FUNCTION_BLOCK ProductOrders (* Basic Function Block Type *)
  (* Standard: 61499-2 *)
  (* Version 0.0, 5/28/2018, taavi, nxtControl GmbH, Template *)
  PACKAGE Main;
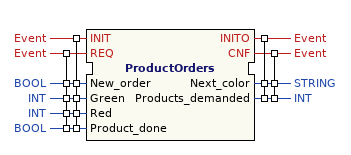
  EVENT_INPUT
    INIT WITH New_order, Green, Red, Product_done; (* Initialization Request *)
    REQ WITH Green, New_order, Product_done, Red; (* Normal Execution Request *)
  END_EVENT
  EVENT_OUTPUT
    INITO WITH Next_color, Products_demanded; (* Initialization Confirm *)
    CNF WITH Next_color, Products_demanded; (* Execution Confirmation *)
  END_EVENT
  VAR_INPUT
    New_order : BOOL;
    Green : INT; (* Input event qualifier *)
    Red : INT;
    Product_done : BOOL;
  END_VAR
  VAR_OUTPUT
    Next_color : STRING; (* Output event qualifier *)
    Products_demanded : INT;
  END_VAR
  VAR
    Green_count : INT;
    Red_count : INT;
    Product_count : INT;
  END_VAR
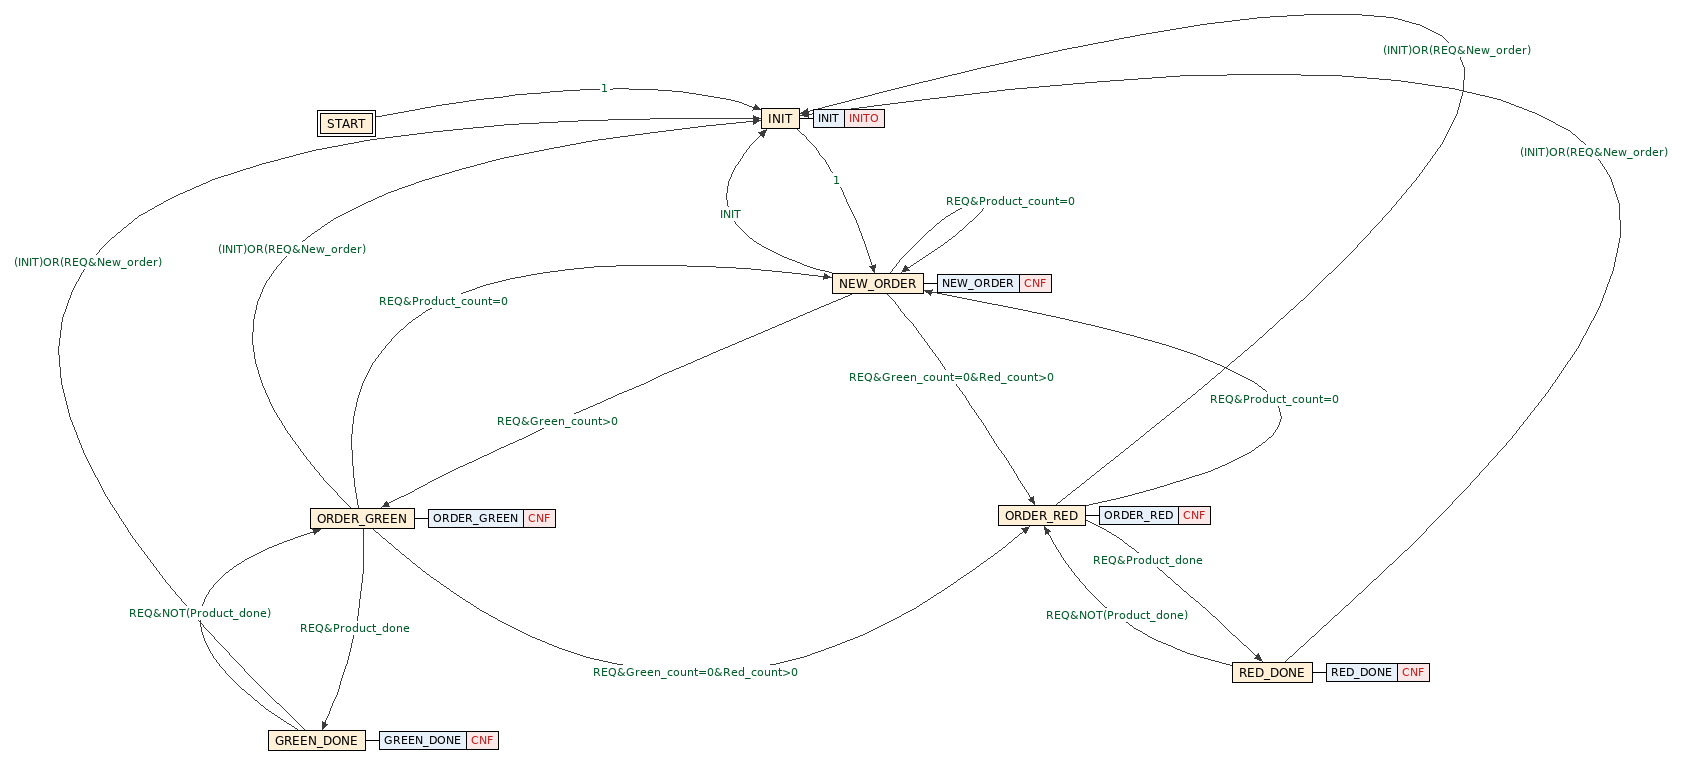
  EC_STATES
    START; (* Initial State *)
    INIT : INIT -> INITO; (* Initialization *)
    NEW_ORDER : NEW_ORDER -> CNF;
    ORDER_GREEN : ORDER_GREEN -> CNF;
    ORDER_RED : ORDER_RED -> CNF;
    GREEN_DONE : GREEN_DONE -> CNF;
    RED_DONE : RED_DONE -> CNF;
  END_STATES
  EC_TRANSITIONS
    START TO INIT := 1;
    INIT TO NEW_ORDER := 1;
    NEW_ORDER TO ORDER_GREEN := REQ&Green_count>0;
    NEW_ORDER TO ORDER_RED := REQ&Green_count=0&Red_count>0;
    NEW_ORDER TO NEW_ORDER := REQ&Product_count=0;
    ORDER_GREEN TO ORDER_RED := REQ&Green_count=0&Red_count>0;
    ORDER_GREEN TO NEW_ORDER := REQ&Product_count=0;
    ORDER_RED TO NEW_ORDER := REQ&Product_count=0;
    ORDER_GREEN TO INIT := (INIT)OR(REQ&New_order);
    ORDER_RED TO INIT := (INIT)OR(REQ&New_order);
    NEW_ORDER TO INIT := INIT;
    ORDER_GREEN TO GREEN_DONE := REQ&Product_done;
    GREEN_DONE TO ORDER_GREEN := REQ&NOT(Product_done);
    ORDER_RED TO RED_DONE := REQ&Product_done;
    RED_DONE TO ORDER_RED := REQ&NOT(Product_done);
    GREEN_DONE TO INIT := (INIT)OR(REQ&New_order);
    RED_DONE TO INIT := (INIT)OR(REQ&New_order);
  END_TRANSITIONS
  ALGORITHM INIT IN ST: (* Initialization algorithm *)
;
Green_count := 0;
Red_count := 0;
Product_count := 0;
Products_demanded := 0;
Next_color := 'NONE';
  END_ALGORITHM
  ALGORITHM NEW_ORDER IN ST:
;
Red_count := Red;
Green_count := Green;
Product_count := Red_count + Green_count;
Products_demanded := Product_count;
Next_color := 'NONE';
  END_ALGORITHM
  ALGORITHM ORDER_GREEN IN ST:
;
Products_demanded := Product_count;
Next_color := 'GREEN';
  END_ALGORITHM
  ALGORITHM ORDER_RED IN ST:
;
Products_demanded := Product_count;
Next_color := 'RED';
  END_ALGORITHM
  ALGORITHM GREEN_DONE IN ST:
;
Green_count := Green_count - 1;
Product_count := Green_count + Red_count;
Products_demanded := Product_count;
Next_color := 'GREEN';
  END_ALGORITHM
  ALGORITHM RED_DONE IN ST:
;
Red_count := Red_count - 1;
Product_count := Green_count + Red_count;
Products_demanded := Product_count;
Next_color := 'RED';
  END_ALGORITHM
END_FUNCTION_BLOCK
